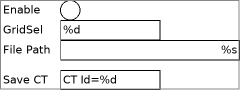
VISUALIZATION _VISU_WorkerDefGrid_VerifyDetail  // 240x90
VAR_IN_OUT
		m_Inst : FB_WorkerDefGrid_Verify;
END_VAR
    Rectangle (60,70 100x20), "CT Id=%d", text variable: m_Inst.nCTId
    Rectangle (60,20 100x20), "%d", text variable: m_Inst.nSelectGridTable
        OnMouseClick: write the text variable via Default
    Rectangle (0,20 60x20), "GridSel"
    Rectangle (0,70 60x20), "Save CT"
    Rectangle (0,0 60x20), "Enable"
    Ellipse (60,0 20x20)
        toggle m_Inst.bEnableGridExport
    Rectangle (60,40 180x20), "%s", text variable: m_Inst.sOutputPath
        OnMouseClick: write the text variable via Default
    Rectangle (0,40 60x20), "File Path"
END_VISUALIZATION

(* stored: Version 1.1.0.1, ProductVersion 3.1.4024.11
   Visu _VISU_WorkerDefGrid_VerifyDetail: Id {02c4b999-e579-4c3a-9689-23d095b68081} *)
